PROGRAM P5_02_DiagramVisualisation
VAR
END_VAR

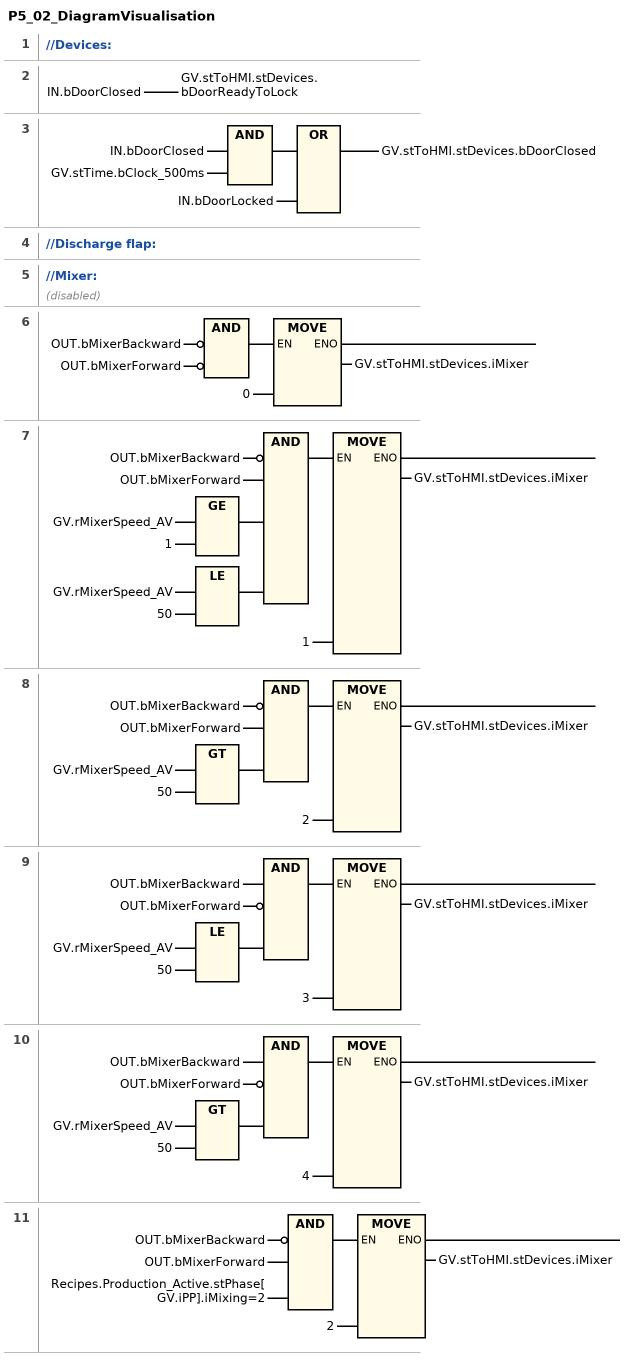
// NETWORK 1
// label: //Devices

// NETWORK 2
GV.stToHMI.stDevices.bDoorReadyToLock := IN.bDoorClosed;

// NETWORK 3
GV.stToHMI.stDevices.bDoorClosed := IN.bDoorClosed AND GV.stTime.bClock_500ms OR IN.bDoorLocked;

// NETWORK 4
// label: //Discharge flap

// NETWORK 5 (disabled)
// label: //Mixer

// NETWORK 6
IF NOT OUT.bMixerBackward AND NOT OUT.bMixerForward THEN GV.stToHMI.stDevices.iMixer := 0; END_IF

// NETWORK 7
IF NOT OUT.bMixerBackward AND OUT.bMixerForward AND GV.rMixerSpeed_AV >= 1 AND GV.rMixerSpeed_AV <= 50 THEN
    GV.stToHMI.stDevices.iMixer := 1;
END_IF

// NETWORK 8
IF NOT OUT.bMixerBackward AND OUT.bMixerForward AND GV.rMixerSpeed_AV > 50 THEN
    GV.stToHMI.stDevices.iMixer := 2;
END_IF

// NETWORK 9
IF OUT.bMixerBackward AND NOT OUT.bMixerForward AND GV.rMixerSpeed_AV <= 50 THEN
    GV.stToHMI.stDevices.iMixer := 3;
END_IF

// NETWORK 10
IF OUT.bMixerBackward AND NOT OUT.bMixerForward AND GV.rMixerSpeed_AV > 50 THEN
    GV.stToHMI.stDevices.iMixer := 4;
END_IF

// NETWORK 11
IF NOT OUT.bMixerBackward AND OUT.bMixerForward AND (Recipes.Production_Active.stPhase[GV.iPP].iMixing=2) THEN
    GV.stToHMI.stDevices.iMixer := 2;
END_IF

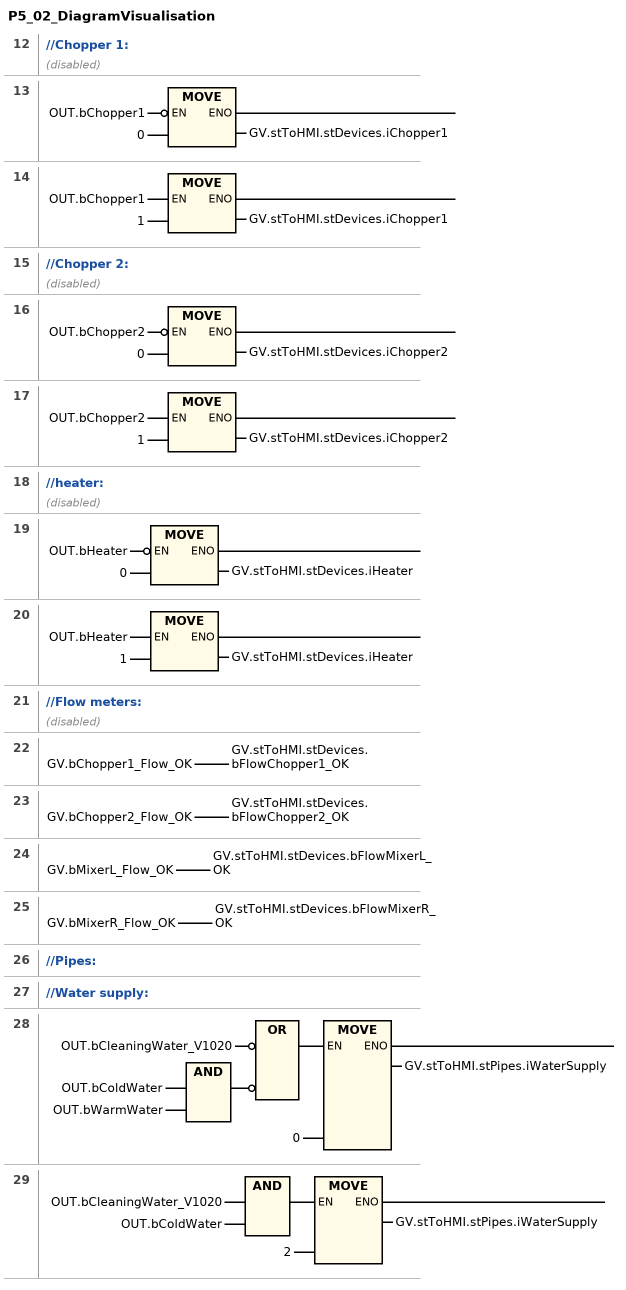
// NETWORK 12 (disabled)
// label: //Chopper 1

// NETWORK 13
IF NOT OUT.bChopper1 THEN GV.stToHMI.stDevices.iChopper1 := 0; END_IF

// NETWORK 14
IF OUT.bChopper1 THEN GV.stToHMI.stDevices.iChopper1 := 1; END_IF

// NETWORK 15 (disabled)
// label: //Chopper 2

// NETWORK 16
IF NOT OUT.bChopper2 THEN GV.stToHMI.stDevices.iChopper2 := 0; END_IF

// NETWORK 17
IF OUT.bChopper2 THEN GV.stToHMI.stDevices.iChopper2 := 1; END_IF

// NETWORK 18 (disabled)
// label: //heater

// NETWORK 19
IF NOT OUT.bHeater THEN GV.stToHMI.stDevices.iHeater := 0; END_IF

// NETWORK 20
IF OUT.bHeater THEN GV.stToHMI.stDevices.iHeater := 1; END_IF

// NETWORK 21 (disabled)
// label: //Flow meters

// NETWORK 22
GV.stToHMI.stDevices.bFlowChopper1_OK := GV.bChopper1_Flow_OK;

// NETWORK 23
GV.stToHMI.stDevices.bFlowChopper2_OK := GV.bChopper2_Flow_OK;

// NETWORK 24
GV.stToHMI.stDevices.bFlowMixerL_OK := GV.bMixerL_Flow_OK;

// NETWORK 25
GV.stToHMI.stDevices.bFlowMixerR_OK := GV.bMixerR_Flow_OK;

// NETWORK 26
// label: //Pipes

// NETWORK 27
// label: //Water supply

// NETWORK 28
IF NOT OUT.bCleaningWater_V1020 OR NOT (OUT.bColdWater AND OUT.bWarmWater) THEN
    GV.stToHMI.stPipes.iWaterSupply := 0;
END_IF

// NETWORK 29
IF OUT.bCleaningWater_V1020 AND OUT.bColdWater THEN GV.stToHMI.stPipes.iWaterSupply := 2; END_IF

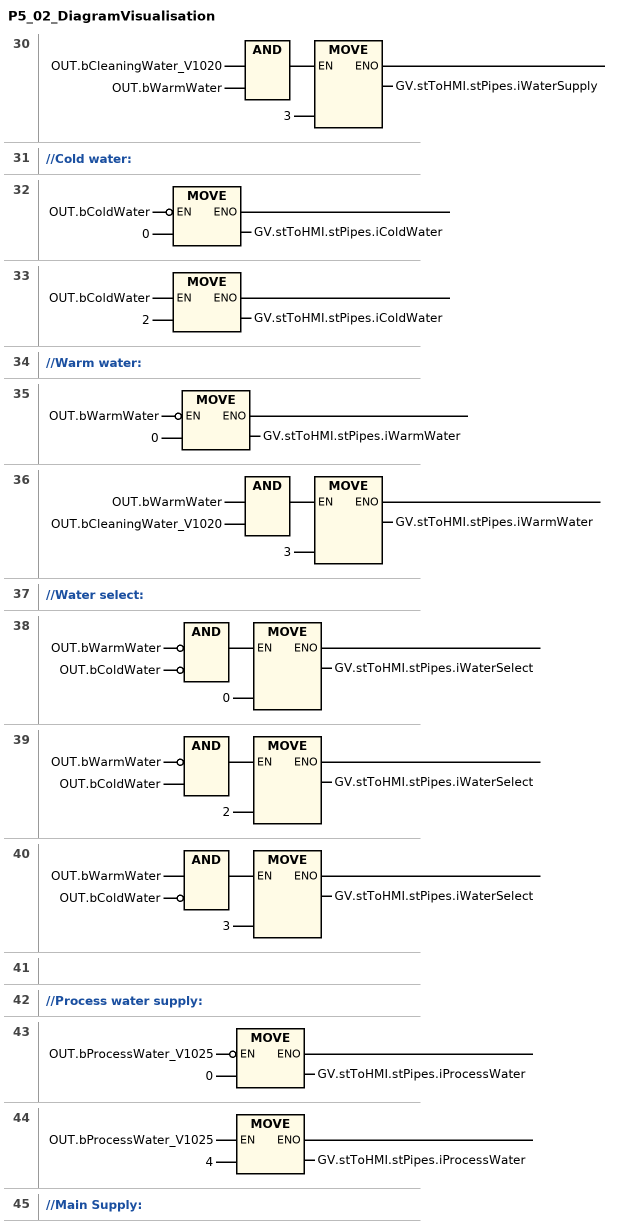
// NETWORK 30
IF OUT.bCleaningWater_V1020 AND OUT.bWarmWater THEN GV.stToHMI.stPipes.iWaterSupply := 3; END_IF

// NETWORK 31
// label: //Cold water

// NETWORK 32
IF NOT OUT.bColdWater THEN GV.stToHMI.stPipes.iColdWater := 0; END_IF

// NETWORK 33
IF OUT.bColdWater THEN GV.stToHMI.stPipes.iColdWater := 2; END_IF

// NETWORK 34
// label: //Warm water

// NETWORK 35
IF NOT OUT.bWarmWater THEN GV.stToHMI.stPipes.iWarmWater := 0; END_IF

// NETWORK 36
IF OUT.bWarmWater AND OUT.bCleaningWater_V1020 THEN GV.stToHMI.stPipes.iWarmWater := 3; END_IF

// NETWORK 37
// label: //Water select

// NETWORK 38
IF NOT OUT.bWarmWater AND NOT OUT.bColdWater THEN GV.stToHMI.stPipes.iWaterSelect := 0; END_IF

// NETWORK 39
IF NOT OUT.bWarmWater AND OUT.bColdWater THEN GV.stToHMI.stPipes.iWaterSelect := 2; END_IF

// NETWORK 40
IF OUT.bWarmWater AND NOT OUT.bColdWater THEN GV.stToHMI.stPipes.iWaterSelect := 3; END_IF

// NETWORK 41

// NETWORK 42
// label: //Process water supply

// NETWORK 43
IF NOT OUT.bProcessWater_V1025 THEN GV.stToHMI.stPipes.iProcessWater := 0; END_IF

// NETWORK 44
IF OUT.bProcessWater_V1025 THEN GV.stToHMI.stPipes.iProcessWater := 4; END_IF

// NETWORK 45
// label: //Main Supply

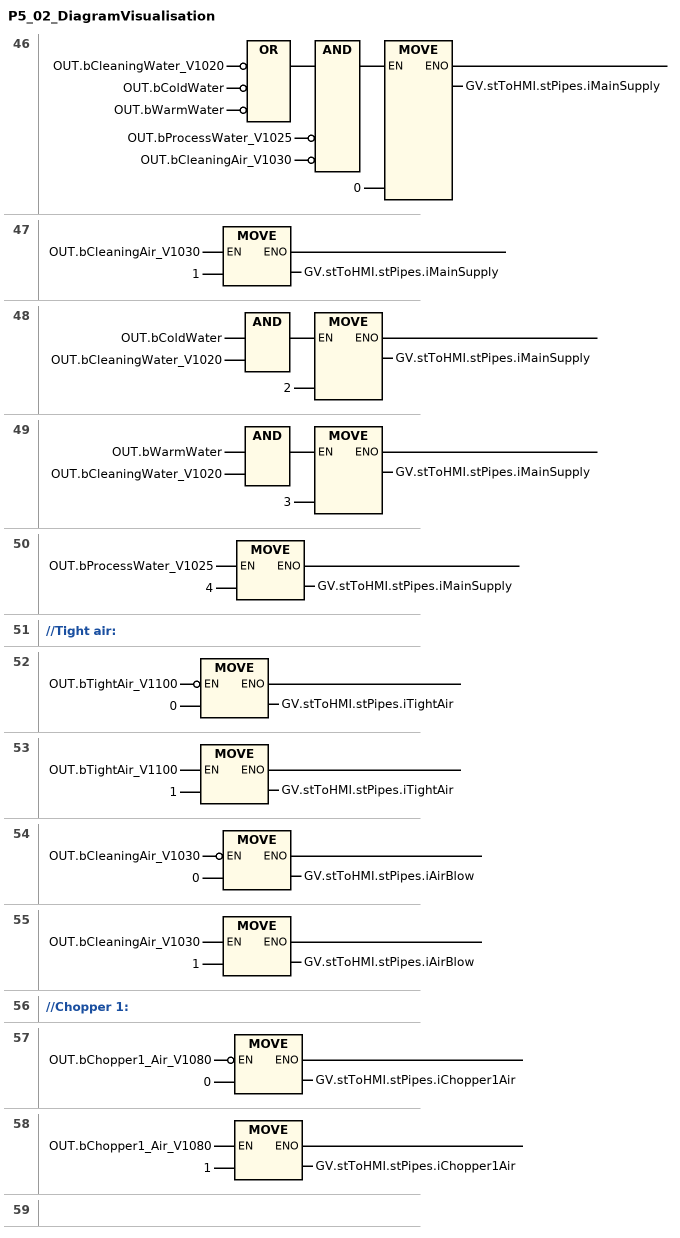
// NETWORK 46
IF (NOT OUT.bCleaningWater_V1020 OR NOT OUT.bColdWater OR NOT OUT.bWarmWater) AND NOT OUT.bProcessWater_V1025 AND NOT OUT.bCleaningAir_V1030 THEN
    GV.stToHMI.stPipes.iMainSupply := 0;
END_IF

// NETWORK 47
IF OUT.bCleaningAir_V1030 THEN GV.stToHMI.stPipes.iMainSupply := 1; END_IF

// NETWORK 48
IF OUT.bColdWater AND OUT.bCleaningWater_V1020 THEN GV.stToHMI.stPipes.iMainSupply := 2; END_IF

// NETWORK 49
IF OUT.bWarmWater AND OUT.bCleaningWater_V1020 THEN GV.stToHMI.stPipes.iMainSupply := 3; END_IF

// NETWORK 50
IF OUT.bProcessWater_V1025 THEN GV.stToHMI.stPipes.iMainSupply := 4; END_IF

// NETWORK 51
// label: //Tight air

// NETWORK 52
IF NOT OUT.bTightAir_V1100 THEN GV.stToHMI.stPipes.iTightAir := 0; END_IF

// NETWORK 53
IF OUT.bTightAir_V1100 THEN GV.stToHMI.stPipes.iTightAir := 1; END_IF

// NETWORK 54
IF NOT OUT.bCleaningAir_V1030 THEN GV.stToHMI.stPipes.iAirBlow := 0; END_IF

// NETWORK 55
IF OUT.bCleaningAir_V1030 THEN GV.stToHMI.stPipes.iAirBlow := 1; END_IF

// NETWORK 56
// label: //Chopper 1

// NETWORK 57
IF NOT OUT.bChopper1_Air_V1080 THEN GV.stToHMI.stPipes.iChopper1Air := 0; END_IF

// NETWORK 58
IF OUT.bChopper1_Air_V1080 THEN GV.stToHMI.stPipes.iChopper1Air := 1; END_IF

// NETWORK 59

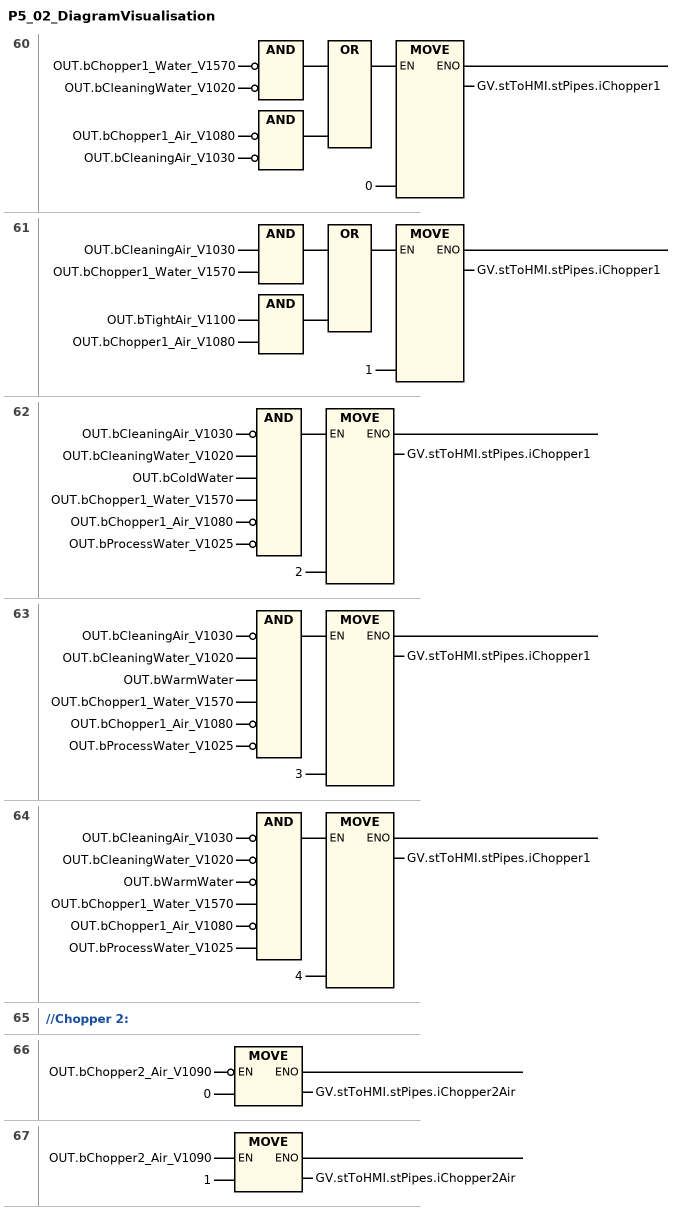
// NETWORK 60
IF NOT OUT.bChopper1_Water_V1570 AND NOT OUT.bCleaningWater_V1020 OR NOT OUT.bChopper1_Air_V1080 AND NOT OUT.bCleaningAir_V1030 THEN
    GV.stToHMI.stPipes.iChopper1 := 0;
END_IF

// NETWORK 61
IF OUT.bCleaningAir_V1030 AND OUT.bChopper1_Water_V1570 OR OUT.bTightAir_V1100 AND OUT.bChopper1_Air_V1080 THEN
    GV.stToHMI.stPipes.iChopper1 := 1;
END_IF

// NETWORK 62
IF NOT OUT.bCleaningAir_V1030 AND OUT.bCleaningWater_V1020 AND OUT.bColdWater AND OUT.bChopper1_Water_V1570 AND NOT OUT.bChopper1_Air_V1080 AND NOT OUT.bProcessWater_V1025 THEN
    GV.stToHMI.stPipes.iChopper1 := 2;
END_IF

// NETWORK 63
IF NOT OUT.bCleaningAir_V1030 AND OUT.bCleaningWater_V1020 AND OUT.bWarmWater AND OUT.bChopper1_Water_V1570 AND NOT OUT.bChopper1_Air_V1080 AND NOT OUT.bProcessWater_V1025 THEN
    GV.stToHMI.stPipes.iChopper1 := 3;
END_IF

// NETWORK 64
IF NOT OUT.bCleaningAir_V1030 AND NOT OUT.bCleaningWater_V1020 AND NOT OUT.bWarmWater AND OUT.bChopper1_Water_V1570 AND NOT OUT.bChopper1_Air_V1080 AND OUT.bProcessWater_V1025 THEN
    GV.stToHMI.stPipes.iChopper1 := 4;
END_IF

// NETWORK 65
// label: //Chopper 2

// NETWORK 66
IF NOT OUT.bChopper2_Air_V1090 THEN GV.stToHMI.stPipes.iChopper2Air := 0; END_IF

// NETWORK 67
IF OUT.bChopper2_Air_V1090 THEN GV.stToHMI.stPipes.iChopper2Air := 1; END_IF

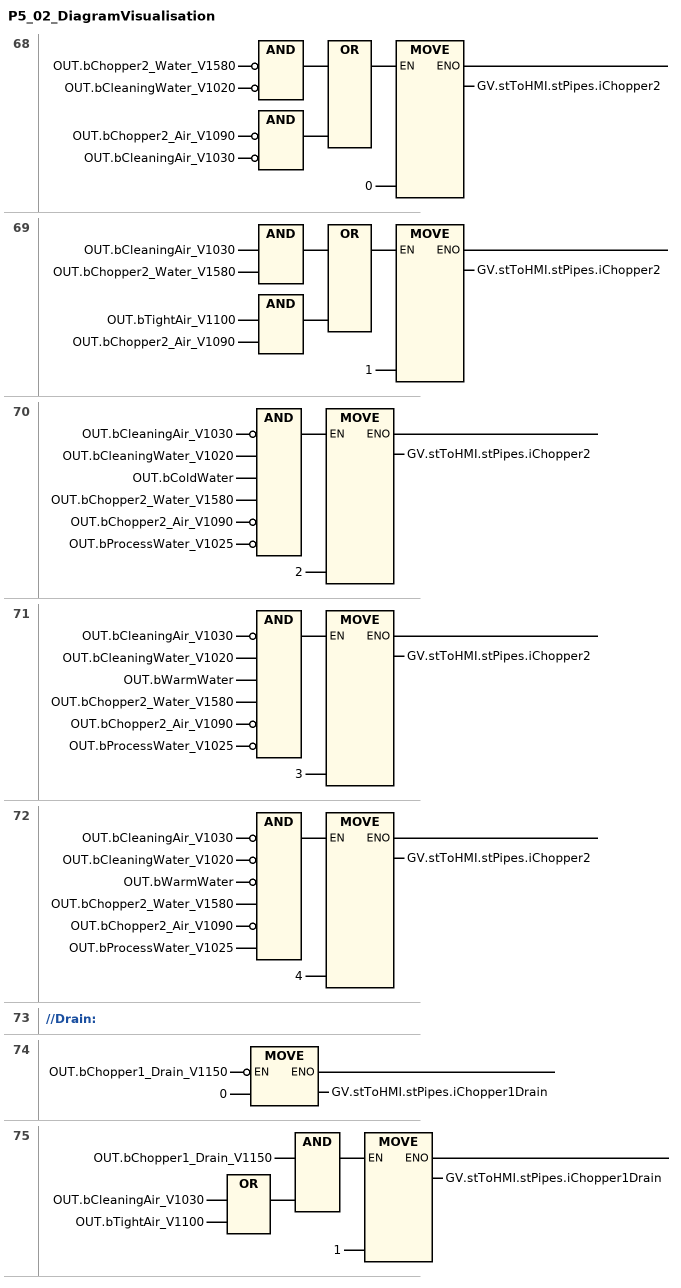
// NETWORK 68
IF NOT OUT.bChopper2_Water_V1580 AND NOT OUT.bCleaningWater_V1020 OR NOT OUT.bChopper2_Air_V1090 AND NOT OUT.bCleaningAir_V1030 THEN
    GV.stToHMI.stPipes.iChopper2 := 0;
END_IF

// NETWORK 69
IF OUT.bCleaningAir_V1030 AND OUT.bChopper2_Water_V1580 OR OUT.bTightAir_V1100 AND OUT.bChopper2_Air_V1090 THEN
    GV.stToHMI.stPipes.iChopper2 := 1;
END_IF

// NETWORK 70
IF NOT OUT.bCleaningAir_V1030 AND OUT.bCleaningWater_V1020 AND OUT.bColdWater AND OUT.bChopper2_Water_V1580 AND NOT OUT.bChopper2_Air_V1090 AND NOT OUT.bProcessWater_V1025 THEN
    GV.stToHMI.stPipes.iChopper2 := 2;
END_IF

// NETWORK 71
IF NOT OUT.bCleaningAir_V1030 AND OUT.bCleaningWater_V1020 AND OUT.bWarmWater AND OUT.bChopper2_Water_V1580 AND NOT OUT.bChopper2_Air_V1090 AND NOT OUT.bProcessWater_V1025 THEN
    GV.stToHMI.stPipes.iChopper2 := 3;
END_IF

// NETWORK 72
IF NOT OUT.bCleaningAir_V1030 AND NOT OUT.bCleaningWater_V1020 AND NOT OUT.bWarmWater AND OUT.bChopper2_Water_V1580 AND NOT OUT.bChopper2_Air_V1090 AND OUT.bProcessWater_V1025 THEN
    GV.stToHMI.stPipes.iChopper2 := 4;
END_IF

// NETWORK 73
// label: //Drain

// NETWORK 74
IF NOT OUT.bChopper1_Drain_V1150 THEN GV.stToHMI.stPipes.iChopper1Drain := 0; END_IF

// NETWORK 75
IF OUT.bChopper1_Drain_V1150 AND (OUT.bCleaningAir_V1030 OR OUT.bTightAir_V1100) THEN
    GV.stToHMI.stPipes.iChopper1Drain := 1;
END_IF

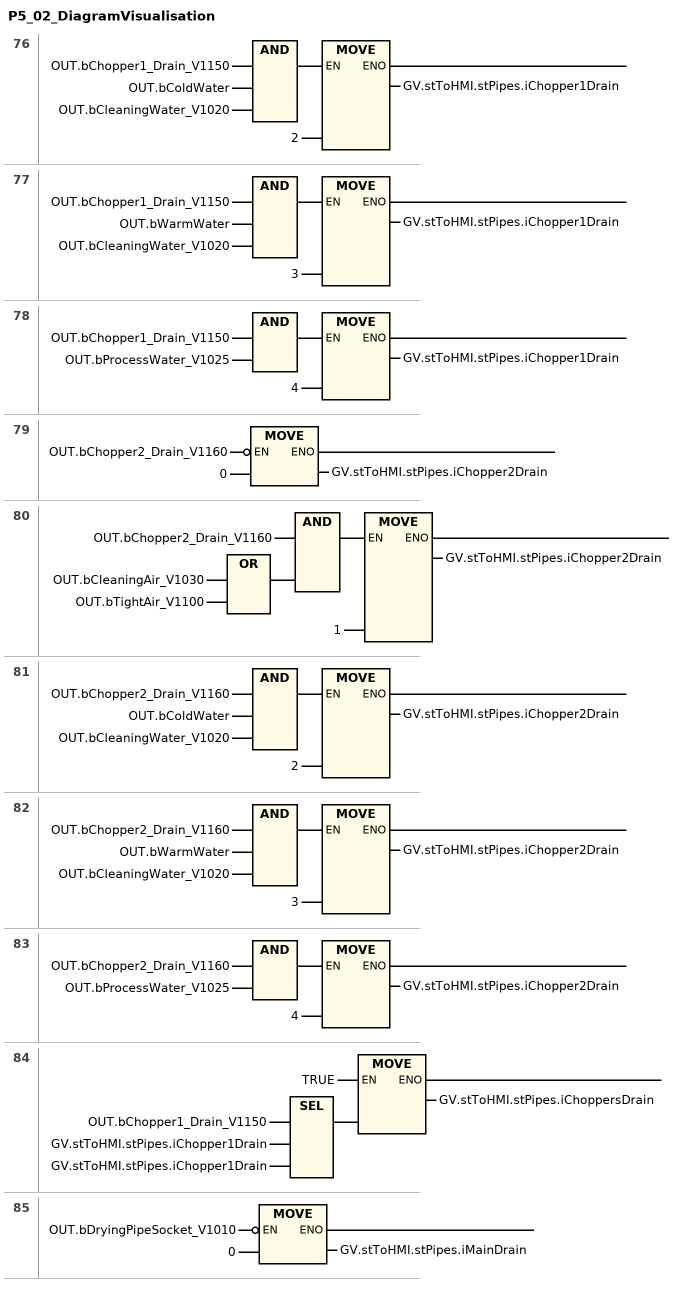
// NETWORK 76
IF OUT.bChopper1_Drain_V1150 AND OUT.bColdWater AND OUT.bCleaningWater_V1020 THEN
    GV.stToHMI.stPipes.iChopper1Drain := 2;
END_IF

// NETWORK 77
IF OUT.bChopper1_Drain_V1150 AND OUT.bWarmWater AND OUT.bCleaningWater_V1020 THEN
    GV.stToHMI.stPipes.iChopper1Drain := 3;
END_IF

// NETWORK 78
IF OUT.bChopper1_Drain_V1150 AND OUT.bProcessWater_V1025 THEN GV.stToHMI.stPipes.iChopper1Drain := 4; END_IF

// NETWORK 79
IF NOT OUT.bChopper2_Drain_V1160 THEN GV.stToHMI.stPipes.iChopper2Drain := 0; END_IF

// NETWORK 80
IF OUT.bChopper2_Drain_V1160 AND (OUT.bCleaningAir_V1030 OR OUT.bTightAir_V1100) THEN
    GV.stToHMI.stPipes.iChopper2Drain := 1;
END_IF

// NETWORK 81
IF OUT.bChopper2_Drain_V1160 AND OUT.bColdWater AND OUT.bCleaningWater_V1020 THEN
    GV.stToHMI.stPipes.iChopper2Drain := 2;
END_IF

// NETWORK 82
IF OUT.bChopper2_Drain_V1160 AND OUT.bWarmWater AND OUT.bCleaningWater_V1020 THEN
    GV.stToHMI.stPipes.iChopper2Drain := 3;
END_IF

// NETWORK 83
IF OUT.bChopper2_Drain_V1160 AND OUT.bProcessWater_V1025 THEN GV.stToHMI.stPipes.iChopper2Drain := 4; END_IF

// NETWORK 84
GV.stToHMI.stPipes.iChoppersDrain := SEL(OUT.bChopper1_Drain_V1150, GV.stToHMI.stPipes.iChopper1Drain, GV.stToHMI.stPipes.iChopper1Drain);

// NETWORK 85
IF NOT OUT.bDryingPipeSocket_V1010 THEN GV.stToHMI.stPipes.iMainDrain := 0; END_IF

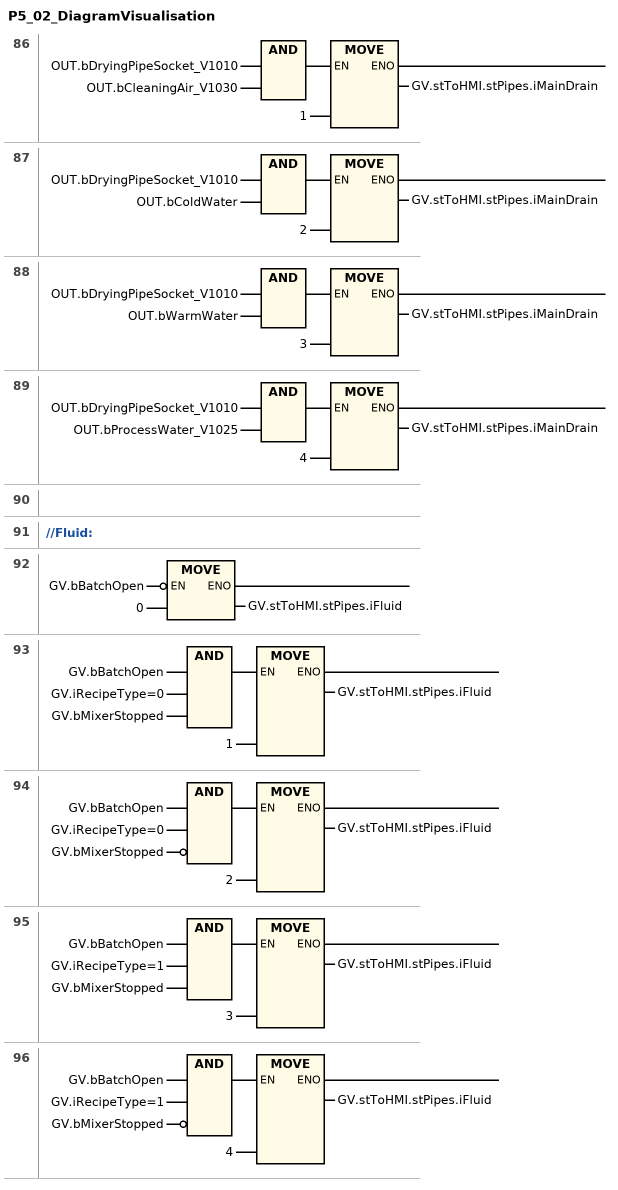
// NETWORK 86
IF OUT.bDryingPipeSocket_V1010 AND OUT.bCleaningAir_V1030 THEN GV.stToHMI.stPipes.iMainDrain := 1; END_IF

// NETWORK 87
IF OUT.bDryingPipeSocket_V1010 AND OUT.bColdWater THEN GV.stToHMI.stPipes.iMainDrain := 2; END_IF

// NETWORK 88
IF OUT.bDryingPipeSocket_V1010 AND OUT.bWarmWater THEN GV.stToHMI.stPipes.iMainDrain := 3; END_IF

// NETWORK 89
IF OUT.bDryingPipeSocket_V1010 AND OUT.bProcessWater_V1025 THEN GV.stToHMI.stPipes.iMainDrain := 4; END_IF

// NETWORK 90

// NETWORK 91
// label: //Fluid

// NETWORK 92
IF NOT GV.bBatchOpen THEN GV.stToHMI.stPipes.iFluid := 0; END_IF

// NETWORK 93
IF GV.bBatchOpen AND (GV.iRecipeType=0) AND GV.bMixerStopped THEN GV.stToHMI.stPipes.iFluid := 1; END_IF

// NETWORK 94
IF GV.bBatchOpen AND (GV.iRecipeType=0) AND NOT GV.bMixerStopped THEN GV.stToHMI.stPipes.iFluid := 2; END_IF

// NETWORK 95
IF GV.bBatchOpen AND (GV.iRecipeType=1) AND GV.bMixerStopped THEN GV.stToHMI.stPipes.iFluid := 3; END_IF

// NETWORK 96
IF GV.bBatchOpen AND (GV.iRecipeType=1) AND NOT GV.bMixerStopped THEN GV.stToHMI.stPipes.iFluid := 4; END_IF

END_PROGRAM

(* stored: Version 1.1.0.1
   POU P5_02_DiagramVisualisation: Id {bc9e8a74-853f-4307-bdae-27c231815e17}, SpecialFunc None *)
